FUNCTION F_FormatString1 : T_MaxString
VAR_INPUT
	Format	: T_MaxString;
	arg1	: T_Arg;
END_VAR
VAR
    FB_FormatString1 : FB_FormatString;
END_VAR

FB_FormatString1(
	sFormat:= Format, 
	arg1:= arg1, 
	arg2:= , 
	arg3:= , 
	arg4:= , 
	arg5:= , 
	arg6:= , 
	arg7:= , 
	arg8:= , 
	arg9:= , 
	arg10:= , 
	bError=> , 
	nErrId=> , 
	sOut=> F_FormatString1);

END_FUNCTION

(* stored: Version 1.1.0.1, ProductVersion 3.1.4024.3
   POU F_FormatString1: Id {43cd74e5-4505-05cc-3eee-5b426f7b4883}, SpecialFunc None *)
